// TIA Portal V19 export
DATA_BLOCK "SinaPara_IDB"   // DB32
// stored: InstanceOfName SinaPara, OfSystemLibElement SinaPara, OfSystemLibVersion 1.1
"SinaPara"
   // VAR_INPUT
   //    Start : Bool;
   //    ReadWrite : Bool;
   //    ParaNo : Int;
   //    AxisNo : Byte;
   //    hardwareId : HW_IO;
   // END_VAR
   // VAR_OUTPUT
   //    Ready : Bool;
   //    Busy : Bool;
   //    Done : Bool;
   //    Error : Bool;
   //    ErrorId : DWord;
   //    DiagId : Word;
   // END_VAR
   // VAR_IN_OUT
   //    Parameter : Array[1..16] of SinaParameter;
   // END_VAR
   // VAR
   //    sbWrError : Bool;
   //    sbWrDone : Bool;
   //    sbRdError : Bool;
   //    sbWrBusy : Bool;
   //    sbRdBusy : Bool;
   //    sbWrStart : Bool;
   //    sbRdStart : Bool;
   //    sbWrStart1 : Bool;
   //    sbRdStart1 : Bool;
   //    sbWrStart2 : Bool;
   //    sbRdStart2 : Bool;
   //    sbStart : Bool;
   //    sbReady : Bool;
   //    sbRead : Bool;
   //    sbWrite : Bool;
   //    sbParaNo : Bool;
   //    sbBusy : Bool;
   //    sbError : Bool;
   //    sbDone : Bool;
   //    siParaNo : Int;
   //    syAxisNo : Byte;
   //    siReqRef : Int;
   //    siErrorId : Int;
   //    siErrorCount : Int;
   //    siMaxErrCount : Int;
   //    swParaError : Word;
   //    sReqParaMulti { S7_SetPoint := 'True'} : SinaReqParaMulti;
   //    sxChaParaMulti { S7_SetPoint := 'True'} : SinaChaParaMulti;
   //    sRespParaMulti { S7_SetPoint := 'True'} : SinaRespParaMulti;
   //    RDREC_1 { S7_SetPoint := 'True'} : RDREC;
   //    WRREC_1 { S7_SetPoint := 'True'} : WRREC;
   //    siParaNoMax : Int;
   //    siLenHeader : Int;
   //    siLenParaMulti : Int;
   //    siLenChaPara : Int;
   // END_VAR
BEGIN
END_DATA_BLOCK
